INTERFACE I_EthercatDiagnosis

// Returns TRUE if an error occurred while performing the scan
PROPERTY Error : BOOL
GET
END_GET
END_PROPERTY

// Gets an array of slaves that have been added to ignore list
PROPERTY IgnoredSlaves : REFERENCE TO ARRAY[0..Tc2_EtherCAT.EC_MAX_SLAVES] OF Tc2_System.T_MaxString
GET
END_GET
END_PROPERTY

// Adds the provided slave to a collection of slaves that will not trigger an error
// Example is slaves that are used on hot connect groups, and when connected should not cause an error. 
METHOD IgnoreSlave
VAR_INPUT
	Name	: Tc2_System.T_MaxString;	// Slave to be ignored if not found or an error is reported back
END_VAR
END_METHOD

// Returns an array of misisng slave names
PROPERTY MissingSlaves : REFERENCE TO ARRAY[0..Tc2_EtherCAT.EC_MAX_SLAVES] OF ST_EthercatSlaveInfo
GET
END_GET
END_PROPERTY

// Reset the internal state machine of diagnosis and clearing any errors, if active.
METHOD Reset
END_METHOD

// Performs a scan on the EtherCAT master, returns TRUE when done.
METHOD Scan	: BOOL
VAR_INPUT
	EcMasterNetId	: AMSNETID;
END_VAR
END_METHOD

// Gets the status based on last executed scan.
PROPERTY Status : E_EthercatDiagnosisStatus
GET
END_GET
END_PROPERTY

END_INTERFACE

(* stored: Version 1.1.0.1, ProductVersion 3.1.4024.14
   Itf I_EthercatDiagnosis: Id {d480e5e2-796f-08c1-2d19-d9a6c0bc5913}
   Property Error: Id {f399f9f6-8a08-073f-31f0-8365faa01d27}
   Get Get: Id {a941b2de-91a5-010d-1db1-4ae5fbd09652}
   Property IgnoredSlaves: Id {582d728a-e4e9-0e33-0a0a-9fcf28b5ab19}
   Get Get: Id {45efd74d-e3fb-019d-01b6-950e28d5a59b}
   Method IgnoreSlave: Id {c0321ce0-8f3e-07e8-07fb-26820061999e}
   Property MissingSlaves: Id {7e540e48-5049-0c72-3a49-fcb1f0bb50f7}
   Get Get: Id {4de20bd8-7b08-0c86-2e67-b4b28be93441}
   Method Reset: Id {88f8dd25-48b3-0f1f-2e79-150016b986a8}
   Method Scan: Id {29224ec9-7a49-0d17-189f-59b55a857805}
   Property Status: Id {fdb7ce96-3bdc-0157-2dc9-65994c8f356b}
   Get Get: Id {9c14e4cf-7339-05e1-29be-64502dd2c40a} *)
